KUKA KRL program: chk_w4_grp3_clo.src

&ACCESS RVO1
&REL 1
&COMMENT Check GRP01 Geschlossen
DEF chk_w4_grp3_clo( )

; Check gripper accelo CLOSE Z3.1/2/3/4/5
;//---- Start User-------

$TIMER[10] = 0
$TIMER_STOP[10] = FALSE

WAIT FOR ($IN[50] AND $IN[52])
WAIT FOR (NOT $IN[49] AND NOT $IN[51])

$TIMER_STOP[10] = TRUE
$TIMER[10] = 0

;//---- End User---------

END
